{attribute 'qualified_only'}
PROGRAM MAIN
VAR
    // Simpele demo: twee schakelaars en een lampje
    // Zet in online mode bSwitch1/bSwitch2 aan/uit en kijk hoe bLamp reageert

    bSwitch1       : BOOL := FALSE;   // Schakelaar 1 (input)
    bSwitch2       : BOOL := FALSE;   // Schakelaar 2 (input)
    bEmergencyStop : BOOL := FALSE;   // Noodstop – forceert lamp uit
    bLamp          : BOOL := FALSE;   // Lamp (output)
END_VAR

// =============================================
// MAIN - Simpele demo met schakelaars en lampje Aidan was hier
// =============================================

// Logica: lamp aan als een van de schakelaars waar is,
// tenzij de noodstop actief is (dan altijd uit)
IF bEmergencyStop THEN
    bLamp := FALSE;
ELSE
    bLamp := bSwitch1 OR bSwitch2;
END_IF;

END_PROGRAM

(* stored: Version 1.1.0.1, ProductVersion 3.5.13.50
   POU MAIN: Id {2dc5b880-9d15-491e-8f3c-929d5ca9c871}, SpecialFunc None *)
